Universal Robots URScript: calibrate_feature.script

#####

speed_move = 0.8
speed_slow = 0.05

kraft_z = 5
kraft_x = 5
kraft_y = 5
max_weg_approach = 0.5
v_z = 0.01
v_x = 0.01
v_y = 0.01


stop_force = 5
apporach_speed = 0.01

def get_edge_point(dir, is_forward_movement):

    speed_vec=[0,0,0,0,0,0]
    if (is_forward_movement == True):
        speed_vec[dir] = apporach_speed
    end
    if (is_forward_movement == False):
        speed_vec[dir] = -apporach_speed
    end

    zero_ftsensor()
    aktforce = get_tcp_force()

	while (norm(aktforce[dir]) < stop_force):
		speedl(speed_vec,0.1,0.05)
		aktforce = get_tcp_force()
	end
    stopl(1)

    pos = get_actual_tcp_pose()

    return pos

end


def calculate_feature(edge1_p1,
                      edge1_p2,
                      edge2_p1,
                      edge2_p2,
                      top_p1,
                      top_p2):

    # ---------------------------------------------------------
    # Erste Kante:
    # Messung durch Bewegung in Basis-X.
    # Die Richtung der Kante ergibt sich aus den beiden
    # Messpositionen.
    # ---------------------------------------------------------

    local line1_dx = edge1_p2[0] - edge1_p1[0]
    local line1_dy = edge1_p2[1] - edge1_p1[1]

    # ---------------------------------------------------------
    # Zweite Kante:
    # Messung durch Bewegung in Basis-Y.
    #
    # Diese Kante wird als X-Achse des neuen Features verwendet.
    # ---------------------------------------------------------

    local line2_dx = edge2_p2[0] - edge2_p1[0]
    local line2_dy = edge2_p2[1] - edge2_p1[1]

    local line1_length = sqrt(
        line1_dx * line1_dx +
        line1_dy * line1_dy
    )

    local line2_length = sqrt(
        line2_dx * line2_dx +
        line2_dy * line2_dy
    )

    # Messpunkte dürfen nicht zu dicht beieinanderliegen
    if (line1_length < 0.01):
        popup(
            "Messpunkte der ersten Kante liegen zu dicht zusammen.",
            title="Kalibrierfehler",
            warning=True,
            error=True,
            blocking=True
        )
        halt
    end

    if (line2_length < 0.01):
        popup(
            "Messpunkte der zweiten Kante liegen zu dicht zusammen.",
            title="Kalibrierfehler",
            warning=True,
            error=True,
            blocking=True
        )
        halt
    end

    # Richtungsvektoren normieren
    line1_dx = line1_dx / line1_length
    line1_dy = line1_dy / line1_length

    line2_dx = line2_dx / line2_length
    line2_dy = line2_dy / line2_length

    # ---------------------------------------------------------
    # Prüfen, ob die Kanten ungefähr rechtwinklig sind
    # ---------------------------------------------------------

    local edge_dot_product = (
        line1_dx * line2_dx +
        line1_dy * line2_dy
    )

    # Bei exakt 90 Grad ist das Skalarprodukt null.
    # 0.15 entspricht ungefähr einer Abweichung von 8.6 Grad.
    if (norm(edge_dot_product) > 0.15):
        popup(
            "Die gemessenen Kanten sind nicht rechtwinklig.",
            title="Kalibrierfehler",
            warning=True,
            error=True,
            blocking=True
        )
        halt
    end

    # ---------------------------------------------------------
    # Schnittpunkt der zwei Geraden berechnen
    #
    # Gerade 1:
    # edge1_p1 + s * line1
    #
    # Gerade 2:
    # edge2_p1 + t * line2
    # ---------------------------------------------------------

    local denominator = (
        line1_dx * line2_dy -
        line1_dy * line2_dx
    )

    if (norm(denominator) < 0.001):
        popup(
            "Die gemessenen Kanten sind nahezu parallel.",
            title="Kalibrierfehler",
            warning=True,
            error=True,
            blocking=True
        )
        halt
    end

    local delta_x = edge2_p1[0] - edge1_p1[0]
    local delta_y = edge2_p1[1] - edge1_p1[1]

    local line1_parameter = (
        delta_x * line2_dy -
        delta_y * line2_dx
    ) / denominator

    local origin_x = (
        edge1_p1[0] +
        line1_parameter * line1_dx
    )

    local origin_y = (
        edge1_p1[1] +
        line1_parameter * line1_dy
    )

    # ---------------------------------------------------------
    # Höhe der Arbeitsfläche
    # ---------------------------------------------------------

    local origin_z = (
        top_p1[2] +
        top_p2[2]
    ) / 2.0

    # ---------------------------------------------------------
    # Winkel der Feature-X-Achse
    #
    # Die zweite Kante definiert die X-Achse.
    # ---------------------------------------------------------

    local feature_angle = atan2(line2_dy, line2_dx)

    # Horizontales Feature:
    # rx = 0
    # ry = 0
    # rz = Drehung um Basis-Z
    local calculated_feature = p[
        origin_x,
        origin_y,
        origin_z,
        0.0,
        0.0,
        feature_angle
    ]

    textmsg("Ursprung X: ", origin_x)
    textmsg("Ursprung Y: ", origin_y)
    textmsg("Ursprung Z: ", origin_z)
    textmsg("Feature-Winkel rad: ", feature_angle)
    textmsg("Feature-Winkel Grad: ", r2d(feature_angle))
    textmsg("Neues Feature: ", calculated_feature)

    return calculated_feature
end


def calibrate_feature():
    home = zp3
    # Kante 1 Messen
    movej(home, a=1.2, v=speed_move)
    movej(measure_point_1, a=1.2, v=speed_move)

    edge_point_1 = get_edge_point(1, True)

    movel(measure_point_1, a=1.2, v=speed_move)
    movel(measure_point_2, a=1.2, v=speed_move)

    edge_point_2 = get_edge_point(1, True)

    movel(measure_point_2, a=1.2, v=speed_move)

    movej(home, a=1.2, v=speed_move)
    movej(zp4, a=1.2, v=speed_move)
    # Kante 2 Messen
    movej(measure_point_3, a=1.2, v=speed_move)

    edge2_point_1 = get_edge_point(0, False)
    movel(measure_point_3, a=1.2, v=speed_move)
    movel(measure_point_4, a=1.2, v=speed_move)

    edge2_point_2 = get_edge_point(0, False)

    movel(measure_point_4, a=1.2, v=speed_move)
    movej(zp4, a=1.2, v=speed_move)
    movej(home, a=1.2, v=speed_move)

    # Höhe Messen
    movel(measure_point_5, a=1.2, v=speed_move)

    top_point_1 = get_edge_point(2, False)

    movel(measure_point_6, a=1.2, v=speed_move)

    top_point_2 = get_edge_point(2, False)

    movej(home, a=1.2, v=speed_move)

    global Feature_cal = calculate_feature(
        edge2_point_1,
        edge2_point_2,
        edge_point_1,
        edge_point_2,
        top_point_1,
        top_point_2
    )

    textmsg("Kalibrierung abgeschlossen.")
    textmsg("Gespeichertes Feature: ", RQS_Werk_ref)
end


calibrate_feature()
